TYPE ST_RAA_6_1_CommandArgs :
STRUCT
	Key			: STRING(SIS_6_1.RAA_COMMAND_ARGS_KEY_STRINGLENGTH); // Key
	Value		: STRING(SIS_6_1.RAA_COMMAND_ARGS_VALUE_STRINGLENGTH); // Value
END_STRUCT
END_TYPE

(* stored: Version 1.1.0.1, ProductVersion 3.1.4022.12
   DUT ST_RAA_6_1_CommandArgs: Id {6247dfed-8684-4b26-9a70-47e991b7afa4} *)
